// TIA Portal V15.1 export
// export: Created 2024-06-21T08:40:55.5761379Z, ExportSetting WithDefaults, DisplayName Totally Integrated Automation Portal, DisplayVersion V15.1 Update 5, DisplayName TIA Portal Openness, DisplayVersion V15.1 Update 5, DisplayName SINAMICS Startdrive Advanced, DisplayVersion V15.1, DisplayName G130, G150, S120, S150, SINAMICS MV, S210, DisplayVersion V15.1, DisplayName G110M, G120, G120C, G120D, G120P, DisplayVersion V15.1, DisplayName STEP 7 Professional, DisplayVersion V15.1 Update 5, DisplayName STEP 7 Safety, DisplayVersion V15.1, DisplayName WinCC Professional, DisplayVersion V15.1 Update 5, DisplayName SIMATIC Visualization Architect, DisplayVersion V15.1
FUNCTION "LAlarmSummaryMerge" : Void   // FC2536, FBD
TITLE = LAlarmSummary / LAlarmSummaryMerge
{ S7_Optimized_Access := 'TRUE' }
VERSION : 0.1
// =============================================================================
// This module is used to sum all alarm's from all objects "FB&FC's" and the send it to LMode & LSystemVar-S71500
// =============================================================================
// =============================================================================
// FC tom merge Alarm UDT's
// Shall be called in last network of  upperlevel -1
// =============================================================================
// stored: AutoNumber false, IsIECCheckEnabled false, SetENOAutomatically False, UDAEnableTagReadback false
   VAR_INPUT
      I_UpperLevelAlarm : "Alarm";   // Alarm UDT Upperlevel
   END_VAR
   VAR_IN_OUT
      IO_Alarm : "Alarm";   // Alarm UDT Upperlevel -1 (1 level under upperlevel)
   END_VAR
BEGIN

NETWORK
TITLE = **** 2.2 - Alarms - Alarm generation **** Alarm's Active
// Alarm's Active
// Activate Alarm A
      A     #I_UpperLevelAlarm.AlarmAActive;
      O     #IO_Alarm.AlarmAActive;
      =     #IO_Alarm.AlarmAActive;

// Activate Alarm B
      A     #I_UpperLevelAlarm.AlarmBActive;
      O     #IO_Alarm.AlarmBActive;
      =     #IO_Alarm.AlarmBActive;

// Activate Alarm C
      A     #I_UpperLevelAlarm.AlarmCActive;
      O     #IO_Alarm.AlarmCActive;
      =     #IO_Alarm.AlarmCActive;

// Activate Alarm D
      A     #I_UpperLevelAlarm.AlarmDActive;
      O     #IO_Alarm.AlarmDActive;
      =     #IO_Alarm.AlarmDActive;

// Activate AlarmABCondition
      A     #I_UpperLevelAlarm.AlarmABCondition;
      O     #IO_Alarm.AlarmABCondition;
      =     #IO_Alarm.AlarmABCondition;
END_FUNCTION
